// TIA Portal project "ref_1516_profinet" (V15.1)
// progetto di riferimento per PLC S7 1516 con bus ProfiNet

(* hardware
DEVICE "S71500/ET200MP station_1"  S7-1500 station
   slot 0: "PM 190W 120/230VAC"  PM 190W 120/230VAC  6EP1333-4BA00
   slot 0: "Telaio di montaggio_0"  Rack  6ES7 590-1***0-0AA0
   slot 1: "PLC_1"  CPU 1516-3 PN/DP  6ES7 516-3AN01-0AB0  V2.6
      slot 3: "Display CPU_1"  6ES7591-1BA00-0AA0
   slot 2: "AI 8xU/I/RTD/TC ST_1"  AI 8xU/I/RTD/TC ST  6ES7 531-7KF00-0AB0  V2.2
   slot 3: "DI 32x24VDC HF_1"  DI 32x24VDC HF  6ES7 521-1BL00-0AB0  V2.1
   slot 4: "AQ 4xU/I ST_1"  AQ 4xU/I ST  6ES7 532-5HD00-0AB0  V2.2
   slot 5: "DQ 32x24VDC/0.5A HF_1"  DQ 32x24VDC/0.5A HF  6ES7 522-1BL01-0AB0  V1.1
DEVICE "ET 200S station_1"  ET 200S station
   slot 0: "Telaio di montaggio_0"  Rail
   slot 0: "IO Device_1_1"  IM 151-3 PN HF  6ES7 151-3BA23-0AB0  V6.1
   slot 1: "PM-E DC24..48V_1"  PM-E 24 to 48VDC  6ES7 138-4CA50-0AB0
   slot 2: "2AI x U ST_1"  2AI x U ST  6ES7 134-4FB01-0AB0
   slot 3: "2AO x U ST_1"  2AO x U ST  6ES7 135-4FB01-0AB0
   slot 4: "2DI x DC24V HF_1"  2DI x 24VDC HF  6ES7 131-4BB01-0AB0
   slot 5: "8DI x DC24V_1"  8DI x 24VDC  6ES7 131-4BF00-0AA0
   slot 6: "PM-E DC24V_1"  PM-E 24VDC  6ES7 138-4CA01-0AA0
   slot 7: "2DO x DC24V / 0,5A HF_1"  2DO x 24VDC / 0.5A HF  6ES7 132-4BB01-0AB0
   slot 8: "2DO x DC24V / 0,5A HF_2"  2DO x 24VDC / 0.5A HF  6ES7 132-4BB01-0AB0
   slot 9: "2DO x DC24V / 0,5A HF_3"  2DO x 24VDC / 0.5A HF  6ES7 132-4BB01-0AB0
   slot 10: "2DO x DC24V / 0,5A HF_4"  2DO x 24VDC / 0.5A HF  6ES7 132-4BB01-0AB0
*)

// ===== PLC "PLC_1"  CPU 1516-3 PN/DP =====

VAR_GLOBAL   // PLC tag table "Tabella delle variabili standard"
   "System_Byte" AT %MB1 : Byte;
   "FirstScan" AT %M1.0 : Bool;
   "DiagStatusUpdate" AT %M1.1 : Bool;
   "AlwaysTRUE" AT %M1.2 : Bool;
   "AlwaysFALSE" AT %M1.3 : Bool;
   "Clock_Byte" AT %MB16383 : Byte;
   "Clock_10Hz" AT %M16383.0 : Bool;
   "Clock_5Hz" AT %M16383.1 : Bool;
   "Clock_2.5Hz" AT %M16383.2 : Bool;
   "Clock_2Hz" AT %M16383.3 : Bool;
   "Clock_1.25Hz" AT %M16383.4 : Bool;
   "Clock_1Hz" AT %M16383.5 : Bool;
   "Clock_0.625Hz" AT %M16383.6 : Bool;
   "Clock_0.5Hz" AT %M16383.7 : Bool;
   "DI0.0" AT %I0.0 : Bool;
   "DI0.1" AT %I0.1 : Bool;
   "DI0.2" AT %I0.2 : Bool;
   "DI0.3" AT %I0.3 : Bool;
   "DI0.4" AT %I0.4 : Bool;
   "DI0.5" AT %I0.5 : Bool;
   "PV1" AT %I0.6 : Bool;
   "PR1" AT %I0.7 : Bool;
   "PV2" AT %I1.0 : Bool;
   "PR2" AT %I1.1 : Bool;
   "JM1" AT %I1.2 : Bool;
   "JM2" AT %I1.3 : Bool;
   "JMA" AT %I1.4 : Bool;
   "JMI" AT %I1.5 : Bool;
   "ACK" AT %I1.6 : Bool;
   "EMERG" AT %I1.7 : Bool;
   "DI2.0" AT %I2.0 : Bool;
   "DI2.1" AT %I2.1 : Bool;
   "a_0" AT %I2.2 : Bool;
   "a_1" AT %I2.3 : Bool;
   "b_0" AT %I2.4 : Bool;
   "b_1" AT %I2.5 : Bool;
   "DI2.6" AT %I2.6 : Bool;
   "DI2.7" AT %I2.7 : Bool;
   "DI3.0" AT %I3.0 : Bool;
   "DI3.1" AT %I3.1 : Bool;
   "DI3.2" AT %I3.2 : Bool;
   "DI3.3" AT %I3.3 : Bool;
   "DI3.4" AT %I3.4 : Bool;
   "DI3.5" AT %I3.5 : Bool;
   "DI3.6" AT %I3.6 : Bool;
   "DI3.7" AT %I3.7 : Bool;
   "DO0.0" AT %Q0.0 : Bool;
   "DO0.1" AT %Q0.1 : Bool;
   "DO0.2" AT %Q0.2 : Bool;
   "DO0.3" AT %Q0.3 : Bool;
   "DO0.4" AT %Q0.4 : Bool;
   "DO0.5" AT %Q0.5 : Bool;
   "DO0.6" AT %Q0.6 : Bool;
   "DO0.7" AT %Q0.7 : Bool;
   "DO1.0" AT %Q1.0 : Bool;
   "DO1.1" AT %Q1.1 : Bool;
   "LV1" AT %Q1.2 : Bool;
   "LR1" AT %Q1.3 : Bool;
   "LV2" AT %Q1.4 : Bool;
   "LR2" AT %Q1.5 : Bool;
   "LACK" AT %Q1.6 : Bool;
   "LSTOP" AT %Q1.7 : Bool;
   "DO2.0" AT %Q2.0 : Bool;
   "DO2.1" AT %Q2.1 : Bool;
   "DO2.2" AT %Q2.2 : Bool;
   "DO2.3" AT %Q2.3 : Bool;
   "DO2.4" AT %Q2.4 : Bool;
   "DO2.5" AT %Q2.5 : Bool;
   "DO2.6" AT %Q2.6 : Bool;
   "DO2.7" AT %Q2.7 : Bool;
   "DO3.0" AT %Q3.0 : Bool;
   "DO3.1" AT %Q3.1 : Bool;
   "DO3.2" AT %Q3.2 : Bool;
   "DO3.3" AT %Q3.3 : Bool;
   "DO3.4" AT %Q3.4 : Bool;
   "DO3.5" AT %Q3.5 : Bool;
   "DO3.6" AT %Q3.6 : Bool;
   "DO3.7" AT %Q3.7 : Bool;
   "POT0" AT %IW4 : Int;
   "POT1" AT %IW6 : Int;
   "AI2" AT %IW8 : Int;
   "AI3" AT %IW10 : Int;
   "AI4" AT %IW12 : Int;
   "AI5" AT %IW14 : Int;
   "AI6" AT %IW16 : Int;
   "AI7" AT %IW18 : Int;
   "AO0" AT %QW4 : Int;
   "AO1" AT %QW6 : Int;
   "AO2" AT %QW8 : Int;
   "AO3" AT %QW10 : Int;
   "YB+" AT %Q13.0 : Bool;
   "YB-" AT %Q13.1 : Bool;
   "YA+" AT %Q12.0 : Bool;
   "YA-" AT %Q12.1 : Bool;
   "FC1" AT %I21.0 : Bool;
   "DO14.0" AT %Q14.0 : Bool;
   "DO14.1" AT %Q14.1 : Bool;
   "DO15.0" AT %Q15.0 : Bool;
   "DO15.1" AT %Q15.1 : Bool;
   "AI8" AT %IW256 : Int;
   "AI9" AT %IW258 : Int;
   "AO4" AT %QW256 : Int;
   "AO5" AT %QW258 : Int;
   "DI21.1" AT %I21.1 : Bool;
   "DI20.0" AT %I20.0 : Bool;
   "DI20.1" AT %I20.1 : Bool;
   "DI20.2" AT %I20.2 : Bool;
   "DI20.3" AT %I20.3 : Bool;
   "DI20.4" AT %I20.4 : Bool;
   "DI20.5" AT %I20.5 : Bool;
   "DI20.6" AT %I20.6 : Bool;
   "DI20.7" AT %I20.7 : Bool;
END_VAR

TYPE "Casella"
   STRUCT
      X : Bool;
      Y : Bool;
      Z : Bool;
   END_STRUCT;
END_TYPE

DATA_BLOCK "Caselle"   // DB1
{ S7_Optimized_Access := 'TRUE' }
VERSION : 0.1
   VAR
      Caselle : Array[0..64] of "Casella";
   END_VAR
BEGIN
END_DATA_BLOCK

FUNCTION_BLOCK "Macchina a Stati"   // FB1, SCL
{ S7_Optimized_Access := 'TRUE' }
VERSION : 0.1
BEGIN
   //Guarda appunti veloci veloci
END_FUNCTION_BLOCK

ORGANIZATION_BLOCK "Main"   // OB1, LAD, ProgramCycle
TITLE = "Main Program Sweep (Cycle)"
{ S7_Optimized_Access := 'TRUE' }
VERSION : 0.1
   VAR_INPUT
      Initial_Call : Bool;   // Initial call of this OB
      Remanence : Bool;   // =True, if remanent data are available
   END_VAR
BEGIN

REGION Network 1
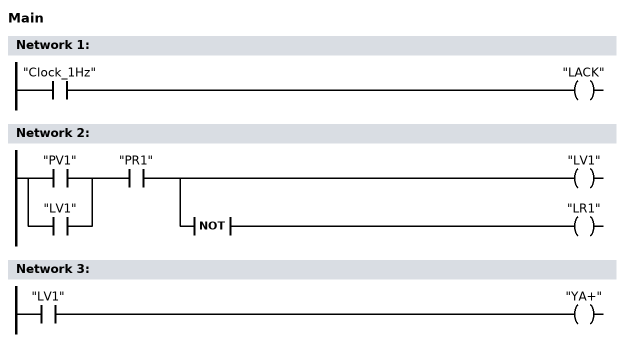
   RUNG wire#powerrail
      Contact( "Clock_1Hz" )
      Coil( "LACK" )
   END_RUNG
   // the same network as SCL:
   "LACK" := "Clock_1Hz";
END_REGION

REGION Network 2
   RUNG wire#powerrail
      Contact( "PV1" )
      wire#w1
      Contact( "PR1" )
      wire#w2
      Coil( "LV1" )
   END_RUNG
   RUNG wire#powerrail
      Contact( "LV1" )
   END_RUNG wire#w1
   RUNG wire#w2
      Not()
      Coil( "LR1" )
   END_RUNG
   // the same network as SCL:
   "LV1" := ("PV1" OR "LV1") AND "PR1";
   "LR1" := NOT "LV1";
END_REGION

REGION Network 3
   RUNG wire#powerrail
      Contact( "LV1" )
      Coil( "YA+" )
   END_RUNG
   // the same network as SCL:
   "YA+" := "LV1";
END_REGION
END_ORGANIZATION_BLOCK